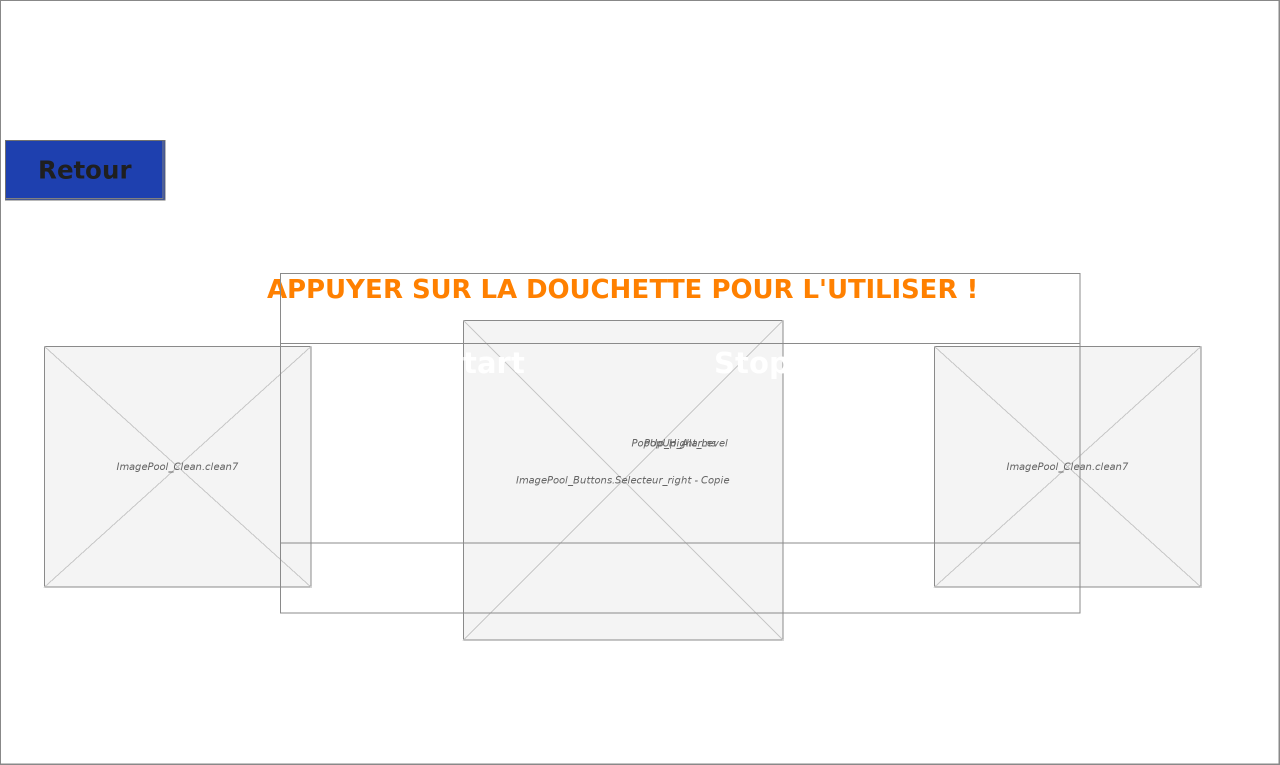
VISUALIZATION Nettoyage  // 1280x765
    Frame (0,0 1280x765)
        shows masque()
    Rectangle (384,706 478x50), "Mesure : %.0f Vol/h", text variable: MES_Debit_Volh_Soufflage
    Group (44,346 267x241)
        Image (0,0 267x241), text variable: NOT GVL_Visu.Cmd_Img_Clean1, invisible if: NOT GVL_Visu.Cmd_Img_Clean1, image: ImagePool_Clean.clean1
        Image (0,0 267x241), text variable: NOT GVL_Visu.Cmd_Img_Clean2, invisible if: NOT GVL_Visu.Cmd_Img_Clean2, image: ImagePool_Clean.clean2
        Image (0,0 267x241), text variable: NOT GVL_Visu.Cmd_Img_Clean3, invisible if: NOT GVL_Visu.Cmd_Img_Clean3, image: ImagePool_Clean.clean3
        Image (0,0 267x241), text variable: NOT GVL_Visu.Cmd_Img_Clean4, invisible if: NOT GVL_Visu.Cmd_Img_Clean4, image: ImagePool_Clean.clean4
        Image (0,0 267x241), text variable: NOT GVL_Visu.Cmd_Img_Clean4, invisible if: NOT GVL_Visu.Cmd_Img_Clean5, image: ImagePool_Clean.clean5
        Image (0,0 267x241), text variable: NOT GVL_Visu.Cmd_Img_Clean6, invisible if: NOT GVL_Visu.Cmd_Img_Clean6, image: ImagePool_Clean.clean6
        Image (0,0 267x241), text variable: NOT GVL_Visu.Cmd_Img_Clean7, invisible if: NOT GVL_Visu.Cmd_Img_Clean7, image: ImagePool_Clean.clean7
    Image (463,320 320x320), invisible if: NOT Start_Etat_Nettoyage, image: ImagePool_Buttons.Selecteur_left
        OnMouseDown: toggle Start_Etat_Nettoyage
    Image (463,320 320x320), invisible if: Start_Etat_Nettoyage, image: ImagePool_Buttons.Selecteur_right - Copie
        OnMouseDown: toggle Start_Etat_Nettoyage
    Rectangle (358,338 170x50), "Start"
    Rectangle (711,338 170x50), "Stop"
    Group (934,346 267x241)
        Image (0,0 267x241), text variable: NOT GVL_Visu.Cmd_Img_Clean1, invisible if: NOT GVL_Visu.Cmd_Img_Clean1, image: ImagePool_Clean.clean1
        Image (0,0 267x241), text variable: NOT GVL_Visu.Cmd_Img_Clean2, invisible if: NOT GVL_Visu.Cmd_Img_Clean2, image: ImagePool_Clean.clean2
        Image (0,0 267x241), text variable: NOT GVL_Visu.Cmd_Img_Clean3, invisible if: NOT GVL_Visu.Cmd_Img_Clean3, image: ImagePool_Clean.clean3
        Image (0,0 267x241), text variable: NOT GVL_Visu.Cmd_Img_Clean4, invisible if: NOT GVL_Visu.Cmd_Img_Clean4, image: ImagePool_Clean.clean4
        Image (0,0 267x241), text variable: NOT GVL_Visu.Cmd_Img_Clean4, invisible if: NOT GVL_Visu.Cmd_Img_Clean5, image: ImagePool_Clean.clean5
        Image (0,0 267x241), text variable: NOT GVL_Visu.Cmd_Img_Clean6, invisible if: NOT GVL_Visu.Cmd_Img_Clean6, image: ImagePool_Clean.clean6
        Image (0,0 267x241), text variable: NOT GVL_Visu.Cmd_Img_Clean7, invisible if: NOT GVL_Visu.Cmd_Img_Clean7, image: ImagePool_Clean.clean7
    Group (139,169 968x144), invisible if: NOT Mode_Cabine_Nettoyage
        Rectangle (160,0 685x48), "MODE NETTOYAGE EN COURS", invisible if: GVL_Visu.On_Off_Anim
        Rectangle (25,48 476x48), "- Vidange(s) ouverte(s)", invisible if: NOT E_Vanne_Vidange_Douche_Ouv
        Rectangle (469,48 476x48), "- Douchette alimentée", invisible if: NOT S_Cmd_Vanne_Alim_Douchette
        Rectangle (0,96 968x48), "APPUYER SUR LA DOUCHETTE POUR L'UTILISER !", invisible if: NOT S_Cmd_Vanne_Alim_Douchette
    RoundedRectangle (412,642 423x65), "Consigne : %.0f Vol/h", text variable: Cons_Deb_Souf_Etat_Nettoyage
        OnMouseDown: write the text variable via VisuDialogs.Numpad, min 0, max 23, format %.0f
    Button (5,140 160x60), "Retour", invisible if: Mode_Cabine_Nettoyage
        OnMouseDown: change screen: menu
    Group (280,273 800x340)
        Frame (0,0 800x340), invisible if: NOT GVL_Visu.Affichage_PopUp_Alarm
            shows PopUp_Alarms()
        Frame (0,70 800x200), invisible if: NOT GVL_Visu.Affichage_PopUp_HightLevel
            shows PopUp_Hight_Level()
END_VISUALIZATION

(* stored: Version 1.1.0.1, ProductVersion 3.1.4024.15
   Visu Nettoyage: Id {01d0c4e2-0a80-475f-91d9-11930f89496c} *)
